{attribute 'qualified_only'}
VAR_GLOBAL
END_VAR

(* stored: Version 1.1.0.1, ProductVersion 3.1.4024.10
   GVL GVL_HMI: Id {53f5ba43-edb6-44b7-b79b-0a21a963890e} *)
